{attribute 'qualified_only'}
VAR_GLOBAL
END_VAR

(* stored: Version 1.1.0.1, ProductVersion 3.1.4024.12
   GVL Itf: Id {62c56635-23ca-4a47-a45b-a51818c30de4} *)
